PROGRAM MAIN
VAR
	(*HXR Accelerator side PLC Interface*)
	{attribute 'TcLinkTo' :=	'TIIB[EBD_E5_EL1008]^Channel 1^Input;
	'}
	i_xUpstreamTreaty_PressOK	AT	%I*	:	BOOL;
	
	{attribute 'TcLinkTo' :=	'TIIB[EBD_E8_EL2794]^Channel 1^Output;
	'}
	q_xUpstreamTreaty_PressOK	AT	%Q*	:	BOOL;
	
	(*HXR Gas Attenuator PLC Interface*)

	(*TXI PLC Interface*)

	(*XPP PLC Interface*)
	
END_VAR

// Run the Diagnostics PRG
DIAGNOSTICS();

(*HXR Accelerator side PLC Interface*)
//Update Accelerator Gauge Pressure Reading
Accelerator_Upstream_Gauge.xPRESS_OK	:=	i_xUpstreamTreaty_PressOK;
//update pressure reading from epics? orsomething?

//Provide Pressure OK reading for Upstream Accelerator Vacuum System
(*
IF  Accelerator_Upstream_Gauge.rPress <= r_Accelerator_Setpoint THEN
	q_xUpstreamTreaty_PressOK	:=	TRUE;
ELSE
	q_xUpstreamTreaty_PressOK	:=	FALSE;
END_IF
*)

(*HXR Gas Attenuator PLC Interface*)

(*TXI PLC Interface*)

(*XPP PLC Interface*)


(*PIRANI Gauges*)

	TV1L0_GPI_01(PG=>);
	
	TV2L0_GPI_01(PG=>);
	
	TV2L0_GPI_02(PG=>);
	
	SL1L0_POWER_GPI_01(PG=>);
	
	AT2L0_SOLID_GPI_01(PG=>);
	
	SP1L0_KMONO_GPI_01(PG=>);
	
	PA1L0_GPI_01(PG=>);
	
	MR1L0_HOMS_GPI_01(PG=>);
	
	MR1L1_TXI_GPI_01(PG=>);
	
	BT2L0_PLEG_GPI_01(PG=>);
	
	MR2L0_HOMS_GPI_01(PG=>);
	
	ST1L0_XTES_GPI_01(PG=>);
	
	(*H1.1 and H1.2
	TV4L0_GPI_01(PG=>);
	
	TV4L0_GPI_02(PG=>);

	TV5L0_GPI_01(PG=>);
	
	TV5L0_GPI_02(PG=>);
	
	*)
	
(*Cold Cathode Gauges*)
	
	TV1L0_GCC_01(PG:=TV1L0_GPI_01.PG,IG=>);
	
	TV2L0_GCC_01(PG:=TV2L0_GPI_01.PG, IG=>);
	
	//TV2L0_GFS_01(PG:=TV2L0_GPI_02.PG,IG=>);
	
	TV2L0_GCC_02(PG:=TV2L0_GPI_02.PG,IG=>);
	
	SL1L0_POWER_GCC_01(PG:=SL1L0_POWER_GPI_01.PG,IG=>);
	
	AT2L0_SOLID_GCC_01(PG:=AT2L0_SOLID_GPI_01.PG,IG=>);
	
	SP1L0_KMONO_GCC_01(PG:=SP1L0_KMONO_GPI_01.PG,IG=>);
	
	PA1L0_GCC_01(PG:=PA1L0_GPI_01.PG,IG=>);
	
	MR1L0_HOMS_GCC_01(PG:=MR1L0_HOMS_GPI_01.PG,IG=>);
	
	MR1L1_TXI_GCC_01(PG:=MR1L1_TXI_GPI_01.PG,IG=>);
	
	BT2L0_PLEG_GCC_01(PG:=BT2L0_PLEG_GPI_01.PG,IG=>);
	
	MR2L0_HOMS_GCC_01(PG:=MR2L0_HOMS_GPI_01.PG,IG=>);
	
	ST1L0_XTES_GCC_01(PG:=ST1L0_XTES_GPI_01.PG,IG=>);

	(*H1.1 and H1.2
	TV4L0_GCC_01(PG:=TV4L0_GPI_01.PG,IG=>);
	
	TV4L0_GCC_02(PG:=TV4L0_GPI_02.PG,IG=>);

	TV5L0_GCC_01(PG:=TV5L0_GPI_01.PG,IG=>);
	
	TV5L0_GCC_02(PG:=TV5L0_GPI_02.PG,IG=>);
	
	TV5L0_GFS_01(PG:=TV5L0_GPI_02.PG,IG=>);

	
	*)
	
	
	
(*Ion Pumps*)

	RTDSL0_PIP_01(i_stGauge:=TV1L0_GCC_01.IG, stPump=>);
	
	RTDSL0_PIP_02(i_stGauge:=TV1L0_GCC_01.IG, stPump=>);
	
	RTDSL0_PIP_03(i_stGauge:=TV1L0_GCC_01.IG, stPump=>);
	
	RTDSL0_PIP_04(i_stGauge:=TV1L0_GCC_01.IG, stPump=>);
	
	RTDSL0_PIP_05(i_stGauge:=TV1L0_GCC_01.IG, stPump=>);
	
	IM1L0_XTES_PIP_01(i_stGauge:=TV2L0_GCC_01.IG, stPump=>);
	
	TV2L0_PIP_01(i_stGauge:=TV2L0_GCC_01.IG, stPump=>);
	
	TV2L0_PIP_02(i_stGauge:=TV2L0_GCC_02.IG, stPump=>);
	
	TV2L0_PIP_03(i_stGauge:=TV2L0_GCC_02.IG, stPump=>);
	
	SL1L0_POWER_PIN_01(i_stGauge:=SL1L0_POWER_GCC_01.IG, stPump=>);
	
	AT2L0_SOLID_PIN_01(i_stGauge:=AT2L0_SOLID_GCC_01.IG, stPump=>);
	
	SP1L0_KMONO_PIP_01(i_stGauge:=SP1L0_KMONO_GCC_01.IG, stPump=>);
	
	PA1L0_PIN_01(i_stGauge:=SP1L0_KMONO_GCC_01.IG, stPump=>); //PIN???	Do I also need CC setpoint?
	
	MR1L0_HOMS_PIP_01(i_stGauge:=MR1L0_HOMS_GCC_01.IG, stPump=>);
	
	MR1L1_TXI_PIP_01(i_stGauge:=MR1L1_TXI_GCC_01.IG, stPump=>);
	
	BT2L0_PLEG_PIP_01(i_stGauge:=BT2L0_PLEG_GCC_01.IG, stPump=>);
	
	MR2L0_HOMS_PIP_01(i_stGauge:=MR2L0_HOMS_GCC_01.IG, stPump=>);
	
	TV3L0_PIP_01(i_stGauge:=ST1L0_XTES_GCC_01.IG, stPump=>);
	
	ST1L0_XTES_PIP_01(i_stGauge:=ST1L0_XTES_GCC_01.IG, stPump=>);
	
	
	(*H1.1 and H1.2
	TV4L0_PIP_01(i_stGauge:=TV4L0_GCC_01.IG, stPump=>);
	
	TV4L0_PIP_02(i_stGauge:=TV4L0_GCC_02.IG, stPump=>);
	
	PA2L0_PIN_01 : FB_PIP_Gamma;
	
	TV5L0_PIP_01(i_stGauge:=TV5L0_GCC_01.IG, stPump=>);
	
	TV5L0_PIP_02(i_stGauge:=TV5L0_GCC_02.IG, stPump=>);
	*)

(*Vacuum Gate Valve*)
	
	TV1L0_VGC_01(
	i_stUSG:= Accelerator_Upstream_Gauge, 
	i_stDSG:= TV1L0_GCC_01.IG, 
	i_xDis_DPIlk:= FALSE , 
	i_xEPS_OK:= TRUE, 
	i_xPMPS_OK:= TRUE, 
	i_xExt_OK:= TRUE, 
	i_xOverrideMode:= xSystemOverrideMode_EBD, 
	i_xReset:= xReset_PMPS_FFO1, 
	iq_stValve=> , 
	xMPS_OK=> , 
	io_fbFFHWO:= g_FastFaultOutput1);
	
	IM1L0_XTES_VGC_01(
	i_stUSG:= TV1L0_GCC_01.IG, 
	i_stDSG:= TV2L0_GCC_01.IG, 
	i_xDis_DPIlk:= FALSE , 
	i_xEPS_OK:= TRUE, 
	i_xPMPS_OK:= TRUE, 
	i_xExt_OK:= TRUE, 
	i_xOverrideMode:= xSystemOverrideMode_EBD, 
	i_xReset:= xReset_PMPS_FFO1, 
	iq_stValve=> , 
	xMPS_OK=> , 
	io_fbFFHWO:= g_FastFaultOutput1);

	TV2L0_VGC_01(
	i_stUSG:= TV2L0_GCC_01.IG, 
	i_stDSG:= TV2L0_GCC_02.IG, 
	i_xDis_DPIlk:= FALSE , 
	i_xEPS_OK:= TRUE, 
	i_xPMPS_OK:= TRUE, 
	i_xExt_OK:= TRUE, 
	i_xOverrideMode:= xSystemOverrideMode_EBD, 
	i_xReset:= xReset_PMPS_FFO1, 
	iq_stValve=> , 
	xMPS_OK=> , 
	io_fbFFHWO:= g_FastFaultOutput1);
	
	TV2L0_VGC_02(
	i_stUSG:= TV2L0_GCC_02.IG, 
	i_stDSG:= SL1L0_POWER_GCC_01.IG, 
	i_xDis_DPIlk:= FALSE , 
	i_xEPS_OK:= TRUE, 
	i_xPMPS_OK:= TRUE, 
	i_xExt_OK:= TRUE, 
	i_xOverrideMode:= xSystemOverrideMode_FEE, 
	i_xReset:= xReset_PMPS_FFO1, 
	iq_stValve=> , 
	xMPS_OK=> , 
	io_fbFFHWO:= g_FastFaultOutput1);
	
	PC1L0_XTES_VGC_01(
	i_stUSG:= AT2L0_SOLID_GCC_01.IG, 
	i_stDSG:= SP1L0_KMONO_GCC_01.IG, 
	i_xDis_DPIlk:= FALSE , 
	i_xEPS_OK:= TRUE, 
	i_xPMPS_OK:= TRUE, 
	i_xExt_OK:= TRUE, 
	i_xOverrideMode:= xSystemOverrideMode_FEE, 
	i_xReset:= xReset_PMPS_FFO1, 
	iq_stValve=> , 
	xMPS_OK=> , 
	io_fbFFHWO:= g_FastFaultOutput1);
	
//	PA1L0_VFS_01 : FB_VFS;

	MR1L0_HOMS_VGC_01(
	i_stUSG:= PA1L0_GCC_01.IG, 
	i_stDSG:= MR1L0_HOMS_PIP_01.q_IG, 
	i_xDis_DPIlk:= FALSE , 
	i_xEPS_OK:= TRUE, 
	i_xPMPS_OK:= TRUE, 
	i_xExt_OK:= TRUE, 
	i_xOverrideMode:= xSystemOverrideMode_FEE, 
	i_xReset:= xReset_PMPS_FFO1, 
	iq_stValve=> , 
	xMPS_OK=> , 
	io_fbFFHWO:= g_FastFaultOutput1);

	BT2L0_PLEG_VGC_01(
	i_stUSG:= MR1L0_HOMS_PIP_01.q_IG, 
	i_stDSG:= BT2L0_PLEG_GCC_01.IG, 
	i_xDis_DPIlk:= FALSE , 
	i_xEPS_OK:= TRUE, 
	i_xPMPS_OK:= TRUE, 
	i_xExt_OK:= TRUE, 
	i_xOverrideMode:= xSystemOverrideMode_FEE, 
	i_xReset:= xReset_PMPS_FFO1, 
	iq_stValve=> , 
	xMPS_OK=> , 
	io_fbFFHWO:= g_FastFaultOutput1);

	MR2L0_HOMS_VGC_01(
	i_stUSG:= BT2L0_PLEG_GCC_01.IG, 
	i_stDSG:= MR2L0_HOMS_GCC_01.IG, 
	i_xDis_DPIlk:= FALSE , 
	i_xEPS_OK:= TRUE, 
	i_xPMPS_OK:= TRUE, 
	i_xExt_OK:= TRUE, 
	i_xOverrideMode:= xSystemOverrideMode_FEE, 
	i_xReset:= xReset_PMPS_FFO1, 
	iq_stValve=> , 
	xMPS_OK=> , 
	io_fbFFHWO:= g_FastFaultOutput1);	
	
	MR2L0_HOMS_VGC_02(
	i_stUSG:= MR2L0_HOMS_GCC_01.IG, 
	i_stDSG:= ST1L0_XTES_GCC_01.IG, 
	i_xDis_DPIlk:= FALSE , 
	i_xEPS_OK:= TRUE, 
	i_xPMPS_OK:= TRUE, 
	i_xExt_OK:= TRUE, 
	i_xOverrideMode:= xSystemOverrideMode_FEE, 
	i_xReset:= xReset_PMPS_FFO1, 
	iq_stValve=> , 
	xMPS_OK=> , 
	io_fbFFHWO:= g_FastFaultOutput1);

	TV1L1_VGC_01(
	i_stUSG:= MR1L1_TXI_GCC_01.IG, 
	i_stDSG:= MR2L0_HOMS_GCC_01.IG, 
	i_xDis_DPIlk:= FALSE , 
	i_xEPS_OK:= TRUE, 
	i_xPMPS_OK:= TRUE, 
	i_xExt_OK:= TRUE, 
	i_xOverrideMode:= xSystemOverrideMode_FEE, 
	i_xReset:= xReset_PMPS_FFO1, 
	iq_stValve=> , 
	xMPS_OK=> , 
	io_fbFFHWO:= g_FastFaultOutput1);		

//	TV3L0_VFS_01 : FB_VFS;

//	PC2L1_L2SI_VGC_01 : FB_VGC;

	(*H1.1
	TV4L0_VGC_01(
	i_stUSG:= TV4L0_GCC_01.IG, 
	i_stDSG:= TV4L0_GCC_02.IG, 
	i_xDis_DPIlk:= FALSE , 
	i_xEPS_OK:= TRUE, 
	i_xPMPS_OK:= TRUE, 
	i_xExt_OK:= TRUE, 
	i_xOverrideMode:= xSystemOverrideMode_H1_1_H1_2, 
	i_xReset:= xReset_PMPS_FFO2, 
	iq_stValve=> , 
	xMPS_OK=> , 
	io_fbFFHWO:= g_FastFaultOutput2);	
	
		
	TV5L0_VGC_01(
	i_stUSG:= TV4L0_GCC_02.IG, 
	i_stDSG:= TV5L0_GCC_01.IG, 
	i_xDis_DPIlk:= FALSE , 
	i_xEPS_OK:= TRUE, 
	i_xPMPS_OK:= TRUE, 
	i_xExt_OK:= TRUE, 
	i_xOverrideMode:= xSystemOverrideMode_H1_1_H1_2, 
	i_xReset:= xReset_PMPS_FFO2, 
	iq_stValve=> , 
	xMPS_OK=> , 
	io_fbFFHWO:= g_FastFaultOutput2);	
		
	TV5L0_VGC_02(
	i_stUSG:= TV5L0_GCC_01.IG, 
	i_stDSG:= TV5L0_GCC_02.IG, 
	i_xDis_DPIlk:= FALSE , 
	i_xEPS_OK:= TRUE, 
	i_xPMPS_OK:= TRUE, 
	i_xExt_OK:= TRUE, 
	i_xOverrideMode:= xSystemOverrideMode_H1_1_H1_2, 
	i_xReset:= xReset_PMPS_FFO2, 
	iq_stValve=> , 
	xMPS_OK=> , 
	io_fbFFHWO:= g_FastFaultOutput2);	
	
	TV6L0_VGC_01(
	i_stUSG:= TV5L0_GCC_02.IG, 
	i_stDSG:= XPP_Downstream_Vacuum, 
	i_xDis_DPIlk:= FALSE , 
	i_xEPS_OK:= TRUE, 
	i_xPMPS_OK:= TRUE, 
	i_xExt_OK:= TRUE, 
	i_xOverrideMode:= xSystemOverrideMode_H1_1_H1_2, 
	i_xReset:= xReset_PMPS_FFO2, 
	iq_stValve=> , 
	xMPS_OK=> , 
	io_fbFFHWO:= g_FastFaultOutput2);		
	*)

(*Vacuum Fast Shutter Valve*)

END_PROGRAM

(* stored: Version 1.1.0.1, ProductVersion 3.1.4022.18
   POU MAIN: Id {53e436ba-9af9-4ca4-ad7b-a6b2399fa417}, SpecialFunc None *)
